FUNCTION_BLOCK REAL2TIME_8 (* Basic Function Block Type *)
  (* Standard: 61499-2 *)
  (* Version 0.0, 6/13/2026, Schneider Electric, Template *)
  PACKAGE SE.Nereda;
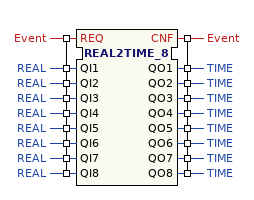
  EVENT_INPUT
    REQ WITH QI1, QI2, QI3, QI4, QI5, QI6, QI7, QI8; (* Normal Execution Request *)
  END_EVENT
  EVENT_OUTPUT
    CNF WITH QO1, QO2, QO3, QO4, QO5, QO6, QO7, QO8; (* Execution Confirmation *)
  END_EVENT
  VAR_INPUT
    QI1 : REAL; (* Input event qualifier *)
    QI2 : REAL;
    QI3 : REAL;
    QI4 : REAL;
    QI5 : REAL;
    QI6 : REAL;
    QI7 : REAL;
    QI8 : REAL;
  END_VAR
  VAR_OUTPUT
    QO1 : TIME; (* Output event qualifier *)
    QO2 : TIME;
    QO3 : TIME;
    QO4 : TIME;
    QO5 : TIME;
    QO6 : TIME;
    QO7 : TIME;
    QO8 : TIME;
  END_VAR
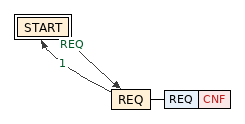
  EC_STATES
    START; (* Initial State *)
    REQ : REQ -> CNF; (* Normal execution *)
  END_STATES
  EC_TRANSITIONS
    START TO REQ := REQ;
    REQ TO START := 1;
  END_TRANSITIONS
  ALGORITHM REQ IN ST: (* Normally executed algorithm *)
;
QO1 := REAL_TO_TIME(QI1*1000 * 60);
QO2 := REAL_TO_TIME(QI2*1000 * 60);
QO3 := REAL_TO_TIME(QI3*1000 * 60);
QO4 := REAL_TO_TIME(QI4*1000 * 60);
QO5 := REAL_TO_TIME(QI5*1000 * 60);
QO6 := REAL_TO_TIME(QI6*1000 * 60);
QO7 := REAL_TO_TIME(QI7*1000 * 60);
QO8 := REAL_TO_TIME(QI8*1000 * 60);
  END_ALGORITHM
END_FUNCTION_BLOCK
